PROGRAM PRG_PLC1
VAR
	ToPLC_X	  AT %Q* : UDINT;
	
	FromPLC2  AT %I*  :UDINT;
	FromPLC3  AT %I*  :UDINT;
END_VAR

F_ConsumeTime(5);
ToPLC_X := (ToPLC_X + 1) MOD 200;

END_PROGRAM

(* stored: Version 1.1.0.1, ProductVersion 3.1.4026.18
   POU PRG_PLC1: Id {008ff7e3-702c-4b23-834b-f8aafcce3fa4}, SpecialFunc None *)
